PROGRAM Feeder
VAR
	bInterlocksOK	:BOOL;
END_VAR
VAR_OUTPUT
	iStep			:UINT;
	iStepTemp		:UINT;
END_VAR

bInterlocksOK := TRUE;

iStepTemp:=iStep;
CASE iStep OF
	0: //Hold
		IF Station.stControl.bRunning THEN
			iStep := 100;
		END_IF
		
	100: //Work
		;
END_CASE
IF NOT bInterlocksOK THEN
	iStep:=iStepTemp;
END_IF

//Control
Station.stAutoCmd.bFeederSTART := F_StepCMP(iStep, 100, 0, 0, 0, 0, 0, 0, 0, 0, 0);

END_PROGRAM

(* stored: Version 1.1.0.1
   POU Feeder: Id {1683f561-a8f4-4ab1-980c-a580769eef6e}, SpecialFunc None *)
